PROGRAM P_Demo_PTIME_TO_TIME
VAR
    tRealValue           : TIME := T#1S500MS; // 模拟 wire 缓冲区中的 TIME 字段
    pTIMEField           : POINTER TO TIME; // 业务侧先算好的字段地址（ADR 或 pBase+nOff）
    bExtractField        : BOOL; // 在线置 TRUE 触发一次解析
    tRealValue_extracted : TIME; // 解析后的副本，供业务逻辑使用
END_VAR

// ============================================================
// Tc2_Utilities.PTIME_TO_TIME 演示程序（FUNCTION）
// ============================================================
// 场景：从一段二进制 wire 缓冲区里按偏移取 TIME 字段（Modbus/CAN/ADS Raw）。
// 价值：替代手写 pField + nOff + ^ 指针算术；一次调用取值，少打错符号。
// 验证：在线写 tRealValue := T#1S500MS；bExtractField := TRUE；
//       下一周期 tRealValue_extracted 应等于 tRealValue。
// ============================================================

// 业务代码通常已经算好字段地址（pBase + 协议偏移）；演示用 ADR 等价
pTIMEField := ADR(tRealValue);

IF bExtractField AND pTIMEField <> 0 THEN
    // 单次完整调用：避免手写 ^ 解引用，统一风格便于和字节序转换串联
    tRealValue_extracted := PTIME_TO_TIME(pTIMEField);
    bExtractField := FALSE;
END_IF;

END_PROGRAM

(* stored: Version 1.1.0.1, ProductVersion 3.1.4024.5
   POU P_Demo_PTIME_TO_TIME: Id {8f9f4844-0f3a-5aa3-9bb2-b91a3b8ae53f}, SpecialFunc None *)
